FUNCTION_BLOCK FeedInfluentLogic_HMI (* Service Interface Function Block Type *)
  (* Standard: 61499-2 *)
  (* Version 0.0, 6/13/2026, Schneider Electric, template *)
  PACKAGE SE.Nereda;
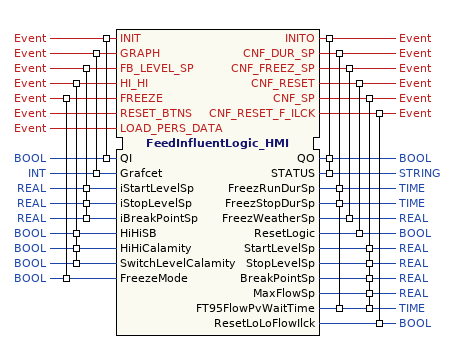
  EVENT_INPUT
    INIT WITH QI;
    GRAPH WITH Grafcet;
    FB_LEVEL_SP WITH iStartLevelSp, iStopLevelSp, iBreakPointSp;
    HI_HI WITH HiHiSB, HiHiCalamity, SwitchLevelCalamity;
    FREEZE WITH FreezeMode;
    RESET_BTNS;
    LOAD_PERS_DATA;
  END_EVENT
  EVENT_OUTPUT
    INITO WITH QO, STATUS;
    CNF_DUR_SP WITH FreezRunDurSp, FreezStopDurSp, FT95FlowPvWaitTime;
    CNF_FREEZ_SP WITH FreezWeatherSp;
    CNF_RESET WITH ResetLogic;
    CNF_SP WITH StartLevelSp, StopLevelSp, BreakPointSp, MaxFlowSp, FT95FlowPvWaitTime;
    CNF_RESET_F_ILCK WITH ResetLoLoFlowIlck;
  END_EVENT
  VAR_INPUT
    QI : BOOL;
    Grafcet : INT;
    iStartLevelSp : REAL;
    iStopLevelSp : REAL;
    iBreakPointSp : REAL;
    HiHiSB : BOOL;
    HiHiCalamity : BOOL;
    SwitchLevelCalamity : BOOL;
    FreezeMode : BOOL;
  END_VAR
  VAR_OUTPUT
    QO : BOOL; (* Event Output Qualifier *)
    STATUS : STRING; (* Service Status *)
    FreezRunDurSp : TIME;
    FreezStopDurSp : TIME;
    FreezWeatherSp : REAL;
    ResetLogic : BOOL;
    StartLevelSp : REAL;
    StopLevelSp : REAL;
    BreakPointSp : REAL;
    MaxFlowSp : REAL;
    FT95FlowPvWaitTime : TIME;
    ResetLoLoFlowIlck : BOOL;
  END_VAR
  SERVICE /
    SEQUENCE 
    END_SEQUENCE
  END_SERVICE
END_FUNCTION_BLOCK
